PROGRAM A_Program
VAR
	i : UINT;

END_VAR

FOR i := 0 TO 100 DO
	B_Program();
END_FOR

END_PROGRAM

(* stored: Version 1.1.0.1, ProductVersion 3.1.4025.12
   POU A_Program: Id {94ff7dcc-e535-4290-85b3-9736c93efdb9}, SpecialFunc None *)
